FUNCTION_BLOCK fBDISCRETE_PID
VAR_INPUT
	Setpoint:REAL;         // SetPoint
    Kp:REAL;               // Kp  Proportional gain
	Ki:REAL;               // Ki  Integrated gain
	Kd:REAL;               // Kd  Derivative gain
	Nfilter:REAL;          // Lowpass Filter Coeff 
	Yprocess :REAL;        // Process Output
	PID_enable : BOOL;     // PId enable (closed loop )
	MV_max_sat : REAL;     // Maximum Saturation
	MV_min_sat : REAL;     // Minimum Saturation
	xExt_Error  :BOOL;     // External error 
END_VAR
VAR_OUTPUT
	MV_out: REAL;
	Inposition:BOOL;     //  4% Settled 
END_VAR
VAR
	T1:DWORD :=0;
	T2:DWORD;
	Perr, Perr1, Perr2 : REAL ;
	A,B,C : REAL;
	prevMV_out:REAL;
	Tsample:REAL;

	pidServo: INT; // Change
END_VAR

//
IF T1 = 0 THEN
	MV_out:=0;     // no bias offset controller
END_IF

Tsample:=0.01;
T1:=REAL_TO_DWORD(Tsample);
Perr:= Setpoint - Yprocess; // Current error e[k]
//
// Constant Coefficients including the Parameters Kp , Ki, Kd and Tsample
//        Your PID Controller algorithm starts here
//

A := (Kp + Ki * (Tsample/2) + (Kd/Tsample));
B := (-Kp + Ki *(Tsample/2) - (2*Kd/Tsample));
C :=  Kd/Tsample;

Mv_out:= prevMV_out +  A*Perr + B * Perr1 + C * Perr2;	// PID Controller
// Instead of old P code
//MV_out:=  Kp * Perr;  // P-Controller

// Update  samples 
prevMV_out := MV_out; // prevMV_out = MV_out[k-1] 
Perr2 := Perr1;       // e[k-2]
Perr1 := Perr;        // e[k-1]



//  PID  is not Enabled 
IF NOT PID_enable THEN
	MV_Out:= Setpoint;
END_IF

//    PID  output saturation 
IF Mv_out < MV_min_sat THEN
	Mv_out:= MV_min_sat;
END_IF
IF Mv_out >  MV_max_sat THEN
	Mv_out:= MV_max_sat;
END_IF
//  PID Output = 0 on External Error <user defined>
IF xExt_Error THEN
	Mv_out:=0;
END_IF

END_FUNCTION_BLOCK

(* stored: Version 1.1.0.1, ProductVersion 3.1.4024.0
   POU fBDISCRETE_PID: Id {6d63eba5-46e9-49ad-b783-0b876d499556}, SpecialFunc None *)
